Yaskawa INFORM job: OK_R2_O38-47,64(2)(90,0)_MPOK.JBI

/JOB
//NAME OK_R2_O38-47,64(2)(90,0)_MPOK
///FOLDERNAME X4
//POS
///NPOS 359,359,359,19,0,0
///TOOL 0
///POSTYPE PULSE
///PULSE
C00000=102904,-190754,-108658,56793,33718,-43054
C00001=112112,-124440,-79629,37912,40591,-30924
C00002=145621,-43895,-45824,14341,74181,-8322
C00003=153971,-33006,-36006,12070,72386,-5523
C00004=154481,-29919,-31590,11999,71202,-5460
C00005=154481,-29717,-30452,12039,70618,-5519
C00006=154481,-29893,-31438,12004,71123,-5468
C00007=153832,-33137,-33612,12213,70898,-5727
C00008=153832,-32934,-32528,12252,70348,-5784
C00009=153968,-31157,-31341,12198,70507,-5716
C00010=153832,-32934,-32528,12252,70348,-5784
C00011=152546,-38024,-38116,12561,71351,-6144
C00012=150032,-44426,-43245,13273,71622,-7027
C00013=145621,-43895,-45824,14341,74181,-8322
C00014=126188,-124725,-79701,29915,35046,-24780
C00015=102904,-190754,-108658,56793,33718,-43054
C00016=131529,-193853,-113060,37345,24088,-27542
C00017=124211,-86804,-80218,19393,77786,-15538
C00018=164541,26866,21690,9198,66417,-2237
C00019=165950,30734,27944,8880,64418,-1868
C00020=167698,37628,37678,8494,61807,-1405
C00021=167698,38233,39472,8555,61023,-1465
C00022=167698,37628,37678,8494,61807,-1405
C00023=167356,33830,33782,8572,62285,-1498
C00024=167337,34588,35914,8650,61376,-1577
C00025=167338,36654,38036,8669,61135,-1595
C00026=167337,34588,35914,8650,61376,-1577
C00027=169007,24634,18452,7731,66783,-560
C00028=157238,-13932,-14846,11323,68842,-4717
C00029=124389,11727,6427,19504,75270,-15913
C00030=120681,54794,37232,20001,79157,-16624
C00031=120183,64187,51861,20385,75351,-17454
C00032=120121,65987,55496,20510,74134,-17689
C00033=120121,66491,57153,20582,73419,-17815
C00034=120121,65987,55496,20510,74134,-17689
C00035=119196,62638,51610,20616,74997,-17884
C00036=119196,63145,53380,20691,74219,-18021
C00037=119742,65256,55831,20631,73685,-17913
C00038=119196,63145,53380,20691,74219,-18021
C00039=119070,39614,17457,20118,83667,-16456
C00040=118481,-15017,-9678,20946,73127,-18482
C00041=136947,-127922,-100425,-9768,37977,-3776
C00042=166532,-153428,-115250,-33739,42272,11545
C00043=160883,-131526,-133102,3483,78120,6366
C00044=103370,-159686,-136025,1765,64172,8056
C00045=97179,-138237,-129333,10238,76593,-11306
C00046=96065,-128281,-122439,10507,77596,-11607
C00047=96065,-128106,-120653,10546,76604,-11690
C00048=96065,-128281,-122439,10507,77596,-11607
C00049=96974,-121186,-120234,10189,79734,-11117
C00050=96065,-128281,-122439,10507,77596,-11607
C00051=80019,-98046,-111669,14399,88698,-15911
C00052=80077,-97852,-111516,14385,88694,-15892
C00053=80077,-98331,-110658,14385,87944,-15982
C00054=80077,-97897,-111441,14385,88627,-15900
C00055=80867,-94680,-110202,14197,89359,-15553
C00056=80077,-97897,-111441,14385,88627,-15900
C00057=77060,-103837,-123440,15157,93336,-16325
C00058=77104,-103620,-123385,15148,93404,-16303
C00059=82212,-117279,-126602,8714,87753,-18646
C00060=83304,-119533,-127995,7425,87342,-19011
C00061=83304,-120285,-126924,7427,86307,-19072
C00062=83304,-120125,-127175,7427,86540,-19060
C00063=84285,-114583,-125380,7184,88184,-18645
C00064=83304,-120125,-127175,7427,86540,-19060
C00065=78124,-131037,-133000,8681,85036,-20864
C00066=78124,-131037,-133000,8681,85036,-20864
C00067=80781,-132367,-131851,8063,83392,-20088
C00068=80781,-132658,-130737,8071,82565,-20142
C00069=80781,-132579,-131090,8068,82820,-20125
C00070=82215,-124520,-128659,7695,85306,-19491
C00071=80136,-136061,-133167,8229,82377,-20371
C00072=80218,-134686,-135534,8183,84509,-20204
C00073=75563,-118157,-129697,13391,92336,-27261
C00074=84024,-123631,-127734,11595,87159,-24981
C00075=84024,-123979,-126960,11598,86516,-25042
C00076=84024,-123746,-127494,11596,86956,-25000
C00077=85048,-122093,-126977,11373,87337,-24623
C00078=81994,-135324,-132084,12059,84184,-25946
C00079=81994,-133752,-136174,12028,87438,-25630
C00080=81994,-133752,-136174,12028,87438,-25630
C00081=83107,-120864,-125937,11789,87596,-25245
C00082=83880,-119254,-122492,11630,86222,-25116
C00083=83880,-119583,-121326,11637,85351,-25197
C00084=83880,-119399,-122020,11633,85865,-25149
C00085=85062,-113328,-120022,11369,87556,-24598
C00086=83880,-119399,-122020,11633,85865,-25149
C00087=83464,-119333,-123502,11716,86850,-25194
C00088=84085,-116294,-122008,11580,87393,-24935
C00089=84085,-116863,-120480,11583,86184,-25047
C00090=84085,-116689,-121008,11580,86590,-25010
C00091=85140,-111307,-119205,11348,88071,-24523
C00092=84085,-116194,-122230,11576,87577,-24918
C00093=82864,-118268,-130611,11862,91757,-24924
C00094=82864,-118268,-130611,11862,91757,-24924
C00095=86851,-110557,-120071,10968,88745,-23893
C00096=86851,-111341,-118540,10968,87421,-24011
C00097=86851,-110811,-119621,10968,88345,-23929
C00098=88598,-109546,-119189,10575,88500,-23337
C00099=86851,-110811,-119621,10968,88345,-23929
C00100=83825,-124590,-131318,11630,88867,-24881
C00101=82909,-127853,-136097,11834,90233,-25054
C00102=84148,-125178,-125504,11579,85018,-25131
C00103=81186,-118241,-121828,12198,86718,-25964
C00104=81186,-118533,-120824,12201,85966,-26037
C00105=81186,-118483,-121017,12200,86107,-26023
C00106=82314,-113243,-119285,11952,87535,-25506
C00107=81186,-118241,-121828,12198,86718,-25964
C00108=87931,-140644,-131144,10841,80108,-24284
C00109=89960,-139833,-128047,10433,78377,-23732
C00110=89960,-139550,-127065,10448,77925,-23770
C00111=89960,-139622,-127307,10444,78035,-23761
C00112=90753,-134395,-125809,10209,79670,-23349
C00113=89456,-143397,-129529,10578,77538,-23979
C00114=95203,-107502,-133483,6717,98684,-21003
C00115=95203,-107502,-133483,6717,98684,-21003
C00116=-70091,-137861,-134613,-19540,89589,11549
C00117=-70091,-137861,-134613,-19540,89589,11549
C00118=-89914,-142582,-130695,-14485,81723,10120
C00119=-90202,-137048,-128128,-14398,82897,9883
C00120=-90202,-136718,-126391,-14423,82025,9985
C00121=-90202,-136862,-127082,-14413,82365,9945
C00122=-91010,-131454,-125503,-14223,83978,9478
C00123=-90202,-137070,-128271,-14397,82970,9874
C00124=-76195,-137070,-128271,-14397,82970,9874
C00125=-74994,-123934,-123423,-14560,86840,9835
C00126=-74994,-124092,-122198,-14564,86029,9931
C00127=-74994,-124005,-122955,-14561,86525,9872
C00128=-76141,-119465,-121513,-14342,87728,9340
C00129=-72631,-133219,-128550,-14998,85696,10781
C00130=-72631,-131663,-134232,-14989,89852,10278
C00131=-50716,-132590,-134806,-14983,95067,21778
C00132=-53786,-122460,-125023,-14607,93736,20890
C00133=-54881,-121663,-124068,-14472,93371,20558
C00134=-54881,-122014,-122728,-14450,92397,20672
C00135=-54881,-121856,-123398,-14460,92875,20616
C00136=-56721,-117465,-121986,-14267,93906,19868
C00137=-54881,-121856,-123398,-14460,92875,20616
C00138=-55322,-120745,-123309,-14420,93300,20415
C00139=-55322,-120747,-123302,-14420,93295,20416
C00140=-55322,-120978,-122461,-14407,92679,20487
C00141=-55322,-120864,-122902,-14414,92999,20450
C00142=-56710,-117554,-121835,-14266,93775,19889
C00143=-54436,-122887,-123768,-14509,92662,20793
C00144=-54436,-122067,-126198,-14556,94519,20574
C00145=-53688,-126302,-127242,-14482,93230,21000
C00146=-7968,-117738,-135568,-14910,102458,19890
C00147=-7968,-117738,-135568,-14910,102458,19890
C00148=-4119,-116606,-125698,-15061,97809,21757
C00149=-7770,-114903,-122318,-14590,96007,20739
C00150=-7770,-115418,-121244,-14557,95111,20843
C00151=-7770,-115024,-122084,-14598,95810,20761
C00152=-9375,-110655,-120613,-14452,96836,20097
C00153=-7770,-115024,-122084,-14598,95810,20761
C00154=-10569,-102485,-118509,-17167,107955,30726
C00155=-17135,-102893,-117262,-17068,107079,30955
C00156=121481,-92648,-105286,5369,115019,86755
C00157=120615,-96829,-107734,5213,114434,86412
C00158=-23859,-150611,-131722,-11614,81196,13147
C00159=-6314,-100679,-115153,-9004,91229,18831
C00160=-5878,-99274,-114584,-9040,91548,18958
C00161=-5881,-109040,-123705,-8960,92007,18939
C00162=-6434,-120006,-133010,-8839,92040,18760
C00163=12667,-120051,-129788,19636,91452,-63850
C00164=15640,-171133,-136982,20070,70138,-66271
C00165=-3139,-164995,-126377,36529,73517,-73495
C00166=120436,-95190,-80290,14692,43277,-16053
C00167=119715,-95468,-78930,15521,42464,-16563
C00168=-536,-140958,-118488,38156,78150,-70805
C00169=15896,-141744,-117960,35334,65109,-67636
C00170=22809,-140005,-116746,30747,58039,-62654
C00171=24043,-118481,-124771,21586,79008,-61529
C00172=24043,-118481,-124771,21586,79008,-61529
C00173=75030,-118005,-124618,21594,79160,-61521
C00174=115715,-153549,-128562,-15788,54400,-49074
C00175=122128,-153495,-122411,-24310,49621,-45021
C00176=120438,-96789,-101713,1489,48968,-3516
C00177=120356,-99154,-104149,1548,49253,-3547
C00178=84431,-115837,-110938,-1908,55230,-61215
C00179=103640,-112319,-105648,-32381,57576,-46168
C00180=90828,-138253,-118809,-13315,45388,-56216
C00181=90828,-138253,-118809,-13315,45388,-56216
C00182=90828,-142934,-129815,-12421,49655,-56806
C00183=90829,-142933,-129813,-12421,49658,-56806
C00184=119872,-163920,-132846,-33283,49576,-42941
C00185=126809,-145866,-124115,-34845,55617,-41735
C00186=120835,-94912,-106201,-4597,84031,-3620
C00187=120296,-100536,-106811,-4468,81494,-3706
C00188=119927,-142522,-122915,-31276,53757,-44413
C00189=77611,-97741,-105288,-5509,51883,-63151
C00190=72401,-92495,-101825,-908,50569,-65138
C00191=77718,-122737,-116129,-5642,44048,-62545
C00192=53268,-154266,-130714,22807,48565,-72872
C00193=53268,-154266,-130714,22807,48565,-72872
C00194=65704,-162398,-123942,17029,37659,-69009
C00195=71918,-162932,-118398,17522,29983,-67437
C00196=120621,-91661,-79831,-4809,93096,80691
C00197=120610,-95504,-82099,-4805,92519,80709
C00198=65560,-150384,-115443,21255,35856,-69819
C00199=55757,-109501,-106397,19317,55331,-70255
C00200=57003,-110782,-106224,17216,52464,-70603
C00201=59740,-113209,-105691,12878,47416,-70775
C00202=50265,-141050,-116073,27906,38980,-77613
C00203=41790,-175398,-134696,41509,59591,-72504
C00204=40096,-167295,-132799,40833,62675,-71982
C00205=66233,-176056,-134792,18069,45461,-58242
C00206=120613,-98309,-97516,18774,58387,-20033
C00207=120296,-100165,-96633,19249,57041,-20409
C00208=66115,-175766,-134726,18105,45590,-58274
C00209=64821,-169609,-132859,18260,47793,-58447
C00210=52681,-139177,-124950,28110,65688,-66537
C00211=50721,-103471,-113434,27126,76369,-64663
C00212=50688,-103205,-113338,27131,76448,-64657
C00213=56284,-114059,-116499,20977,66017,-65546
C00214=54527,-104423,-113142,21374,69156,-65613
C00215=49750,-132075,-132074,23871,68057,-67633
C00216=51888,-141517,-135531,28423,71943,-65142
C00217=58410,-142164,-121837,32385,67064,-69630
C00218=59671,-133628,-117738,33640,70981,-70965
C00219=120621,-92022,-79948,5717,93324,87803
C00220=120611,-95871,-82213,5711,92744,87773
C00221=92104,-176981,-128268,-2909,38154,-41832
C00222=76594,-127084,-115767,-3536,56171,-41355
C00223=99425,-103206,-107694,-29386,75495,-21963
C00224=100715,-115554,-120696,-29641,77391,-21955
C00225=99511,-125054,-130815,-29118,78165,-22610
C00226=-30978,-142903,-136378,-16839,87530,25088
C00227=-49033,-141162,-127974,-10600,82449,19659
C00228=120514,-92773,-72492,-63824,26217,40707
C00229=122096,-91517,-72885,-63277,27653,40461
C00230=-46723,-132150,-125263,-10235,84639,20316
C00231=-38144,-96146,-111322,-6693,87070,23612
C00232=-37356,-92674,-109966,-6904,88077,23811
C00233=-38688,-150385,-135608,-6755,74185,24124
C00234=-34744,-121097,-133452,-9828,92546,23976
C00235=-92930,-150385,-135608,-6755,74185,24124
C00236=-108565,-138971,-125572,-2320,72996,18698
C00237=120610,-93305,-77258,-53115,31058,-22991
C00238=120294,-94166,-75974,-54567,30127,-22239
C00239=-116035,-135916,-124846,7405,75208,6894
C00240=-75325,-100736,-113015,-4102,85156,20630
C00241=-87779,-91378,-109906,9606,90211,4845
C00242=-92139,-118134,-128268,12138,88585,1394
C00243=-96790,-150711,-134355,17072,70659,-2161
C00244=-96790,-150711,-134355,17072,70659,-2161
C00245=-652,-114254,-134536,4800,91191,3391
C00246=166532,-153428,-115250,-33739,42272,11545
C00247=166532,-153428,-115250,-33739,42272,11545
C00248=124114,-84683,-61597,48557,28871,52530
C00249=120971,1491,10647,53300,28999,53238
C00250=122160,19295,36771,64461,24491,47841
C00251=122378,23552,43589,68524,23503,45877
C00252=120673,10502,19535,54974,28515,52685
C00253=120213,7916,15945,54003,29309,53162
C00254=117639,31595,51593,71855,26327,43764
C00255=117542,21645,38109,65998,27616,46690
C00256=116582,-33548,-30911,47449,36332,56383
C00257=108749,-129529,-72544,82443,35289,33776
C00258=107659,-149780,-91003,80990,36184,34408
C00259=234701,-24447,-54419,-57638,71697,-57534
C00260=192045,-4471,-49137,-31395,56880,-70337
C00261=158835,26744,-30866,6797,89214,-71249
C00262=162394,21957,-27190,-640,114363,-79561
C00263=164064,23195,-19161,-1804,117838,-80318
C00264=164490,20804,-18265,-1733,116068,-80136
C00265=164232,27876,-3751,-4961,127378,-83177
C00266=164200,29818,-583,-4904,126429,-83142
C00267=163648,20652,-18364,-1809,116035,-80437
C00268=163648,20933,-18885,-1817,116499,-80445
C00269=162721,21060,-18767,-1901,116472,-80776
C00270=162825,20781,-18263,-1883,116024,-80730
C00271=161869,20798,-18246,-1969,116003,-81071
C00272=161869,21389,-19316,-1987,116965,-81088
C00273=162128,7432,-36637,578,111538,-80469
C00274=155887,-31466,-65010,7215,96475,-81562
C00275=162590,-38859,-73812,1668,81223,-78508
C00276=179792,32070,-16354,-13350,79915,-65662
C00277=186878,-39073,-38836,-41246,34970,-63358
C00278=187458,-25431,-34231,-31791,43871,-67525
C00279=188256,-32514,-32154,-43117,35074,-62369
C00280=188651,-34827,-34931,-42941,35654,-62475
C00281=186634,-25994,-34626,-31183,43526,-67848
C00282=186634,-26042,-35404,-30940,43918,-67999
C00283=179776,-30769,-38597,-15117,38446,-76230
C00284=179862,-30379,-37602,-15341,38064,-76107
C00285=178691,-31104,-38049,-14184,37759,-76698
C00286=185299,-29135,-41036,-26782,46455,-69327
C00287=188726,-40923,-42933,-41373,37038,-63352
C00288=196569,5763,-30645,-36969,53415,-67065
C00289=234701,-24447,-54419,-57638,71697,-57534
C00290=149956,-140196,-108889,10254,17658,75195
C00291=133880,-29999,-59672,20958,46846,70848
C00292=133880,-29999,-59672,20958,46846,70848
C00293=122391,19095,38576,70751,31293,46770
C00294=123405,34197,53895,59777,34432,53030
C00295=120673,9158,15746,60306,37604,52768
C00296=120213,7880,15913,61361,37506,52152
C00297=128224,26945,46555,56859,32016,55120
C00298=125984,18051,32799,53129,35607,56921
C00299=127465,-31665,-25778,42614,42048,63033
C00300=111364,-124873,-96714,53393,47795,55834
C00301=154186,-159927,-117173,847,12331,79725
C00302=85861,-99082,-105113,44329,59147,50836
C00303=83984,-106882,-107996,46165,58479,49488
C00304=120674,-14372,-36148,15341,86455,69375
C00305=120676,-10921,-33498,15340,86592,69392
C00306=125651,22057,-6379,9907,105287,72561
C00307=121175,-12454,-34682,15229,86445,69544
C00308=120675,-14159,-37235,15335,87207,69469
C00309=127950,19387,-8926,9965,105208,73352
C00310=120676,-11639,-34054,15340,86566,69391
C00311=120674,-14390,-36162,15341,86455,69375
C00312=120676,-14354,-36134,15765,85734,-14225
C00313=120676,-14354,-36134,15765,85734,-14225
C00314=121459,-13803,-34784,15590,85060,-14040
C00315=120676,-14158,-37234,15757,86484,-14129
C00316=120165,-16255,-37568,15883,85739,-14397
C00317=124003,-16979,-37218,14998,84465,-13252
C00318=120676,-14374,-36149,15765,85733,-14224
C00319=120676,-14373,-36148,15765,85733,-14225
C00320=98406,-95981,-107671,30899,65126,-25478
C00321=97498,-103141,-110365,31836,63713,-26282
C00322=97498,-103141,-110365,31836,63713,-26282
C00323=151185,-64492,-56891,27025,41971,76525
C00324=173123,2305,9538,10200,51383,-14399
C00325=173123,2305,9538,10200,51383,-14399
C00326=174903,14820,25056,9713,48090,-13953
C00327=177435,27097,40637,4614,49072,-8771
C00328=187315,39588,15664,-2886,77004,-72543
C00329=187570,37474,12233,-2951,78037,-72481
C00330=182393,31000,44587,2257,48438,-6634
C00331=178652,16834,25077,3801,53300,-8079
C00332=172335,1396,7152,6372,56784,-10488
C00333=165460,10359,17772,9398,55625,-13216
C00334=160953,16615,26241,11506,54240,-15214
C00335=161039,26979,37798,10163,56196,-14889
C00336=187825,35310,11263,-3318,76749,7758
C00337=187564,37491,12251,-3232,77251,7657
C00338=166034,27602,38530,8404,55496,-12935
C00339=166237,17707,23738,7975,59455,-12552
C00340=164665,16592,22700,-1550,58461,-2398
C00341=168038,24831,35842,-7675,55527,4086
C00342=167355,24747,35761,-7424,55472,3814
C00343=168052,14770,21803,-7392,58972,3848
C00344=169021,11489,3544,7471,65997,66244
C00345=151185,-64492,-56891,27025,41971,76525
C00346=139846,-133648,-87236,40448,26560,70293
C00347=136335,-97157,-88666,6240,65884,69249
C00348=141826,-62430,-72987,3929,73707,71532
C00349=140052,-21130,-52867,-24635,78479,75610
C00350=128083,45376,-375,-18819,101882,68514
C00351=126763,43366,-45,-18530,100432,68297
C00352=126966,41908,238,-18497,99599,68497
C00353=135984,107314,69748,-14048,119719,69614
C00354=135785,103774,66356,-14147,119946,69504
C00355=122863,47542,6419,-17829,97882,67372
C00356=124413,47820,3838,-18170,99852,67599
C00357=123183,-7178,-53151,6497,97844,73056
C00358=89230,-40025,-45988,57168,55507,51535
BC00000=155259,430035,251707
BC00001=155259,370518,251707
BC00002=155259,370518,251707
BC00003=155259,370518,251707
BC00004=155259,370518,251707
BC00005=155259,370518,251707
BC00006=155259,370518,251707
BC00007=155259,370518,251707
BC00008=155259,370518,251707
BC00009=155259,370518,251707
BC00010=155259,370518,251707
BC00011=155259,370518,251707
BC00012=155259,370518,251707
BC00013=155259,370518,251707
BC00014=155259,370518,251707
BC00015=155259,430035,251707
BC00016=334621,427363,453529
BC00017=334621,347923,356901
BC00018=334621,347923,326221
BC00019=334621,347923,326221
BC00020=334621,347923,326221
BC00021=334621,347923,326221
BC00022=334621,347923,326221
BC00023=334621,347923,326221
BC00024=334621,347923,326221
BC00025=334621,347923,326221
BC00026=334621,347923,326221
BC00027=334621,347923,326221
BC00028=334621,347923,326221
BC00029=334621,347923,326221
BC00030=324461,347923,240729
BC00031=324461,347923,240729
BC00032=324461,347923,240729
BC00033=324461,347923,240729
BC00034=324461,347923,240729
BC00035=324461,347923,240729
BC00036=324461,347923,240729
BC00037=324461,347923,240729
BC00038=324461,347923,240729
BC00039=324461,347923,240729
BC00040=324461,347923,382261
BC00041=343276,399368,267274
BC00042=343276,522663,1074774
BC00043=343276,475512,1074774
BC00044=343276,247728,1074774
BC00045=336018,234000,1074774
BC00046=336018,234000,1074774
BC00047=336018,234000,1074774
BC00048=336018,234000,1074774
BC00049=336018,234000,1074774
BC00050=336018,234000,1074774
BC00051=336018,234000,1074774
BC00052=336018,234000,1074774
BC00053=336018,234000,1074774
BC00054=336018,234000,1074774
BC00055=336018,234000,1074774
BC00056=336018,234000,1074774
BC00057=336018,234000,1074774
BC00058=371484,186454,1072332
BC00059=371484,178806,1072332
BC00060=371484,177238,1072332
BC00061=371484,177238,1072332
BC00062=371484,177238,1072332
BC00063=371484,177238,1072332
BC00064=371484,177238,1072332
BC00065=371484,177238,1072332
BC00066=310125,182966,1071793
BC00067=310125,182966,1071793
BC00068=310125,182966,1071793
BC00069=310125,182966,1071793
BC00070=310125,182966,1071793
BC00071=310125,182966,1071793
BC00072=310125,182966,1071793
BC00073=246912,213302,1071793
BC00074=246912,213302,1071793
BC00075=246912,213302,1071793
BC00076=246912,213302,1071793
BC00077=246912,213302,1071793
BC00078=246912,213302,1071793
BC00079=246912,213302,1071793
BC00080=143996,226029,1063218
BC00081=143996,226029,1063218
BC00082=143996,226029,1063218
BC00083=143996,226029,1063218
BC00084=143996,226029,1063218
BC00085=143996,226029,1063218
BC00086=143996,226029,1063218
BC00087=107402,233101,1063218
BC00088=107402,233101,1063218
BC00089=107402,233101,1063218
BC00090=107402,233101,1063218
BC00091=107402,233101,1063218
BC00092=107402,233101,1063218
BC00093=107402,233101,1063218
BC00094=126000,290967,1063218
BC00095=126000,290967,1063218
BC00096=126000,290967,1063218
BC00097=126000,290967,1063218
BC00098=126000,290967,1063218
BC00099=126000,290967,1063218
BC00100=126000,290967,1063218
BC00101=32367,290967,1063218
BC00102=33707,241035,1063218
BC00103=33707,241035,1063218
BC00104=33707,241035,1063218
BC00105=33707,241035,1063218
BC00106=33707,241035,1063218
BC00107=33707,241035,1063218
BC00108=7031,245739,1063218
BC00109=6955,243723,1064247
BC00110=6955,243723,1064247
BC00111=6955,243723,1064247
BC00112=6955,243723,1064247
BC00113=6955,243723,1064247
BC00114=6955,243723,1064247
BC00115=25087,359545,1064247
BC00116=1824,213285,1064247
BC00117=1824,167485,1064247
BC00118=1824,167485,1064247
BC00119=1824,167485,1064247
BC00120=1824,167485,1064247
BC00121=1824,167485,1064247
BC00122=1824,167485,1064247
BC00123=1824,167485,1064247
BC00124=32224,168989,1065766
BC00125=32224,168989,1065766
BC00126=32224,168989,1065766
BC00127=32224,168989,1065766
BC00128=32224,168989,1065766
BC00129=32224,168989,1065766
BC00130=32224,168989,1065766
BC00131=75962,188381,1065766
BC00132=75961,188380,1065763
BC00133=75961,188380,1065763
BC00134=75961,188380,1065763
BC00135=75961,188380,1065763
BC00136=75961,188380,1065763
BC00137=75961,188380,1065763
BC00138=117533,188380,1065763
BC00139=117533,188380,1065763
BC00140=117533,188380,1065763
BC00141=117533,188380,1065763
BC00142=117533,188380,1065763
BC00143=117533,188380,1065763
BC00144=117533,188380,1065763
BC00145=56658,153797,1065859
BC00146=56658,153797,1065859
BC00147=30873,87130,1065859
BC00148=45198,87130,1065859
BC00149=45198,87130,1065859
BC00150=45198,87130,1065859
BC00151=45198,87131,1065856
BC00152=45198,87131,1065856
BC00153=45198,87131,1065856
BC00154=45198,87131,1065853
BC00155=45198,87131,1065852
BC00156=145241,272408,1075139
BC00157=145241,272408,1075139
BC00158=45198,87131,1065851
BC00159=45198,87131,1065851
BC00160=45198,87131,1065851
BC00161=45198,87131,1065851
BC00162=45198,87131,1065851
BC00163=50333,237173,1065851
BC00164=50333,237173,1065851
BC00165=50333,237173,1065851
BC00166=156919,411124,1075139
BC00167=156919,411124,1075139
BC00168=50333,237173,1065851
BC00169=72120,237173,1065851
BC00170=72120,237173,1065851
BC00171=72120,237173,1065851
BC00172=58630,250517,1065851
BC00173=17,309807,1065851
BC00174=17,261367,1065849
BC00175=17,261367,1065849
BC00176=369303,316629,1075139
BC00177=369303,316629,1075139
BC00178=17,261367,1065849
BC00179=17,261367,1065849
BC00180=17,261367,1065849
BC00181=17,263287,1072219
BC00182=17,340739,1070027
BC00183=271547,213230,1070026
BC00184=312655,207246,1064979
BC00185=312655,207246,1064979
BC00186=4070,330706,1075139
BC00187=4070,330706,1075139
BC00188=312655,207246,1064979
BC00189=312655,207246,1064979
BC00190=312655,207246,1064979
BC00191=312655,207246,1064979
BC00192=312655,207246,1064979
BC00193=280580,230258,1064979
BC00194=280580,230258,1064979
BC00195=280580,230258,1064979
BC00196=125976,418809,1075139
BC00197=125976,418809,1075139
BC00198=280580,230258,1064979
BC00199=280580,230258,1064976
BC00200=280580,230258,1064977
BC00201=280581,230257,1064979
BC00202=280580,230258,1064979
BC00203=280580,230258,1064979
BC00204=211671,216434,1064979
BC00205=204230,216434,1064979
BC00206=168817,338507,1075139
BC00207=168817,338507,1075139
BC00208=204230,216434,1064979
BC00209=204230,216434,1064979
BC00210=204230,216434,1064979
BC00211=204230,216434,1064979
BC00212=204230,216434,1064979
BC00213=204230,216434,1064979
BC00214=204230,216434,1064979
BC00215=204230,216434,1064979
BC00216=93787,231658,1064979
BC00217=93787,231658,1064979
BC00218=93788,231658,1064978
BC00219=27652,419064,1075139
BC00220=27652,419064,1075139
BC00221=93788,231658,1064978
BC00222=93788,231658,1064978
BC00223=93788,231658,1064978
BC00224=93788,231658,1064978
BC00225=93788,231658,1064978
BC00226=58883,202583,1068082
BC00227=58883,202583,1068082
BC00228=345487,351087,1075139
BC00229=345487,351087,1075139
BC00230=58883,202583,1068082
BC00231=58883,202583,1068082
BC00232=58883,202583,1068082
BC00233=58883,202583,1068082
BC00234=58123,202583,1068180
BC00235=1968,161247,1068082
BC00236=1968,161247,1068082
BC00237=310134,354281,1075139
BC00238=310134,354281,1075139
BC00239=1968,161247,1068082
BC00240=1968,161247,1068082
BC00241=1968,161247,1068082
BC00242=1968,161247,1068082
BC00243=1968,161247,1068082
BC00244=1968,356313,1068082
BC00245=56320,430883,1064743
BC00246=343276,475512,1074774
BC00247=343276,475512,418626
BC00248=326702,360123,309424
BC00249=326065,355687,311834
BC00250=325331,353932,278401
BC00251=325331,353932,278401
BC00252=322890,348232,200536
BC00253=322890,348232,200536
BC00254=325331,353932,278401
BC00255=325331,353932,278401
BC00256=325331,353932,278401
BC00257=326702,394520,413552
BC00258=326702,482298,413552
BC00259=301892,455031,17
BC00260=301892,455031,17
BC00261=209904,428615,17
BC00262=165530,382080,91459
BC00263=159566,375826,103748
BC00264=159566,375826,103748
BC00265=146818,362457,130017
BC00266=146818,362457,130017
BC00267=159566,375826,103748
BC00268=159566,375826,103748
BC00269=159566,375826,103748
BC00270=159566,375826,103748
BC00271=159566,375826,103748
BC00272=159566,375826,103748
BC00273=159566,375826,103748
BC00274=160331,376239,102936
BC00275=179623,386657,82465
BC00276=243106,413945,27916
BC00277=213965,383877,85097
BC00278=213965,383877,85097
BC00279=213965,383877,85097
BC00280=213965,383877,85097
BC00281=213965,383877,85097
BC00282=213965,383877,85097
BC00283=213965,383877,85097
BC00284=213965,383877,85097
BC00285=213965,383877,85097
BC00286=213965,383877,85097
BC00287=213965,383877,85097
BC00288=301892,455031,17
BC00289=301892,455031,17
BC00290=376045,502685,343368
BC00291=326979,388611,268695
BC00292=326979,388611,268695
BC00293=314569,362038,322228
BC00294=314569,362038,322228
BC00295=310726,355002,200377
BC00296=310726,355002,200377
BC00297=314569,362038,322228
BC00298=314569,362038,322228
BC00299=314569,362038,322228
BC00300=314569,409194,450098
BC00301=326003,483358,319355
BC00302=108142,501291,133069
BC00303=94929,415794,32572
BC00304=131923,388713,210323
BC00305=131318,389042,183541
BC00306=131077,389173,172829
BC00307=131077,389173,172829
BC00308=131077,389173,172829
BC00309=131077,389173,172829
BC00310=125260,392440,183541
BC00311=125864,392111,210322
BC00312=132288,390101,176526
BC00313=128864,385756,157610
BC00314=127495,384018,150044
BC00315=127495,384018,150044
BC00316=127495,384018,150044
BC00317=127495,384018,150044
BC00318=122392,389386,157610
BC00319=125816,393731,176526
BC00320=132288,412747,17
BC00321=132288,502680,17
BC00322=329813,502680,230019
BC00323=341603,346180,231132
BC00324=341603,346182,356182
BC00325=319069,341990,356182
BC00326=319069,341990,356182
BC00327=319069,341990,385359
BC00328=340757,346640,193638
BC00329=340757,346640,193638
BC00330=319069,341990,385359
BC00331=319069,341990,385359
BC00332=319069,341990,385359
BC00333=319464,342064,382925
BC00334=319464,342064,382925
BC00335=319464,342064,382925
BC00336=344822,337105,170856
BC00337=344822,337105,170856
BC00338=319464,342064,382925
BC00339=319464,342064,382925
BC00340=319464,342064,382925
BC00341=319464,342064,382925
BC00342=319464,342064,382925
BC00343=319464,342064,382925
BC00344=325489,344287,327316
BC00345=341603,346180,395974
BC00346=341603,460199,530170
BC00347=190885,461337,170893
BC00348=190885,404072,170893
BC00349=164847,397070,131538
BC00350=148987,398107,68956
BC00351=148987,398107,68956
BC00352=148987,398107,68956
BC00353=192995,397070,17
BC00354=192995,397070,17
BC00355=148987,398107,68956
BC00356=148987,398107,68956
BC00357=146579,399402,81875
BC00358=106846,403091,165317
EC00000=-798156,-183832
EC00001=-798156,-183832
EC00002=-798156,-183832
EC00003=-798156,-183832
EC00004=-798156,-183832
EC00005=-798156,-183832
EC00006=-798156,-183832
EC00007=-798156,-183832
EC00008=-798156,-183832
EC00009=-798156,-183832
EC00010=-798156,-183832
EC00011=-798156,-183832
EC00012=-798156,-183832
EC00013=-798156,-183832
EC00014=-798156,-183832
EC00015=-798156,-183832
EC00016=-798156,-183832
EC00017=-798156,-183832
EC00018=-798156,-183832
EC00019=-798156,-183832
EC00020=-798156,-183832
EC00021=-798156,-183832
EC00022=-798156,-183832
EC00023=-798156,-183832
EC00024=-798156,-183832
EC00025=-798156,-183832
EC00026=-798156,-183832
EC00027=-798156,-183832
EC00028=-798156,-183832
EC00029=-798156,-183832
EC00030=-798156,-183832
EC00031=-798156,-183832
EC00032=-798156,-183832
EC00033=-798156,-183832
EC00034=-798156,-183832
EC00035=-798156,-183832
EC00036=-798156,-183832
EC00037=-798156,-183832
EC00038=-798156,-183832
EC00039=-798156,-183832
EC00040=-798156,-183832
EC00041=-798156,-183832
EC00042=-798156,-183832
EC00043=-798156,-183832
EC00044=-798156,-183832
EC00045=-798156,-183832
EC00046=-798156,-183832
EC00047=-798156,-183832
EC00048=-798156,-183832
EC00049=-798156,-183832
EC00050=-798156,-183832
EC00051=-798156,-183832
EC00052=-798156,-183832
EC00053=-798156,-183832
EC00054=-798156,-183832
EC00055=-798156,-183832
EC00056=-798156,-183832
EC00057=-798156,-183832
EC00058=-798156,-183832
EC00059=-798156,-183832
EC00060=-798156,-183832
EC00061=-798156,-183832
EC00062=-798156,-183832
EC00063=-798156,-183832
EC00064=-798156,-183832
EC00065=-798156,-183832
EC00066=-798156,-183832
EC00067=-798156,-183832
EC00068=-798156,-183832
EC00069=-798156,-183832
EC00070=-798156,-183832
EC00071=-798156,-183832
EC00072=-798156,-183832
EC00073=-798156,-183832
EC00074=-798156,-183832
EC00075=-798156,-183832
EC00076=-798156,-183832
EC00077=-798156,-183832
EC00078=-798156,-183832
EC00079=-798156,-183832
EC00080=-798156,-183832
EC00081=-798156,-183832
EC00082=-798156,-183832
EC00083=-798156,-183832
EC00084=-798156,-183832
EC00085=-798156,-183832
EC00086=-798156,-183832
EC00087=-798156,-183832
EC00088=-798156,-183832
EC00089=-798156,-183832
EC00090=-798156,-183832
EC00091=-798156,-183832
EC00092=-798156,-183832
EC00093=-798156,-183832
EC00094=-798156,-183832
EC00095=-798156,-183832
EC00096=-798156,-183832
EC00097=-798156,-183832
EC00098=-798156,-183832
EC00099=-798156,-183832
EC00100=-798156,-183832
EC00101=-798156,-183832
EC00102=-798156,-183832
EC00103=-798156,-183832
EC00104=-798156,-183832
EC00105=-798156,-183832
EC00106=-798156,-183832
EC00107=-798156,-183832
EC00108=-798156,-183832
EC00109=-798156,-183832
EC00110=-798156,-183832
EC00111=-798156,-183832
EC00112=-798156,-183832
EC00113=-798156,-183832
EC00114=-798156,-183832
EC00115=-798156,-183832
EC00116=-798156,-183832
EC00117=-798156,-183832
EC00118=-798156,-183832
EC00119=-798156,-183832
EC00120=-798156,-183832
EC00121=-798156,-183832
EC00122=-798156,-183832
EC00123=-798156,-183832
EC00124=-798156,-183832
EC00125=-798156,-183832
EC00126=-798156,-183832
EC00127=-798156,-183832
EC00128=-798156,-183832
EC00129=-798156,-183832
EC00130=-798156,-183832
EC00131=-798156,-183832
EC00132=-798154,-183832
EC00133=-798154,-183832
EC00134=-798154,-183832
EC00135=-798154,-183832
EC00136=-798154,-183832
EC00137=-798154,-183832
EC00138=-798154,-183832
EC00139=-798154,-183832
EC00140=-798154,-183832
EC00141=-798154,-183832
EC00142=-798154,-183832
EC00143=-798154,-183832
EC00144=-798154,-183832
EC00145=-799965,-183832
EC00146=-799965,-183832
EC00147=-799965,-183832
EC00148=-799965,-183832
EC00149=-799965,-183832
EC00150=-799965,-183832
EC00151=-799962,-183833
EC00152=-799962,-183833
EC00153=-799962,-183833
EC00154=-799960,-183834
EC00155=-799958,-183835
EC00156=-975524,-183832
EC00157=-975524,-183832
EC00158=-799958,-183834
EC00159=-799958,-183834
EC00160=-799958,-183834
EC00161=-799958,-183834
EC00162=-799958,-183834
EC00163=-799958,-183834
EC00164=-799958,-183834
EC00165=-799958,-183834
EC00166=-975524,-183832
EC00167=-975524,-183832
EC00168=-799958,-183834
EC00169=-799958,-183834
EC00170=-799958,-183834
EC00171=-799958,-183834
EC00172=-799958,-183834
EC00173=-799958,-183834
EC00174=-799955,-183834
EC00175=-799955,-183834
EC00176=-975524,-183832
EC00177=-975524,-183832
EC00178=-799955,-183834
EC00179=-799955,-183834
EC00180=-799955,-183834
EC00181=-799955,-183834
EC00182=-799954,-183835
EC00183=-799951,-183835
EC00184=-799951,-183835
EC00185=-799951,-183835
EC00186=-975524,-183832
EC00187=-975524,-183832
EC00188=-799951,-183835
EC00189=-799951,-183835
EC00190=-799951,-183835
EC00191=-799951,-183835
EC00192=-799951,-183835
EC00193=-799951,-183835
EC00194=-799951,-183835
EC00195=-799951,-183835
EC00196=-975524,-183832
EC00197=-975524,-183832
EC00198=-799951,-183835
EC00199=-799949,-183836
EC00200=-799950,-183836
EC00201=-799948,-183837
EC00202=-799951,-183835
EC00203=-799951,-183835
EC00204=-799951,-183835
EC00205=-799951,-183835
EC00206=-975524,-183832
EC00207=-975524,-183832
EC00208=-799951,-183835
EC00209=-799951,-183835
EC00210=-799951,-183835
EC00211=-799951,-183835
EC00212=-799951,-183835
EC00213=-799951,-183835
EC00214=-799951,-183835
EC00215=-799951,-183835
EC00216=-799951,-183835
EC00217=-799951,-183835
EC00218=-799949,-183835
EC00219=-975524,-183832
EC00220=-975524,-183832
EC00221=-799949,-183835
EC00222=-799949,-183835
EC00223=-799949,-183835
EC00224=-799949,-183835
EC00225=-799949,-183835
EC00226=-799949,-183835
EC00227=-799949,-183835
EC00228=-975524,-183832
EC00229=-975524,-183832
EC00230=-799949,-183835
EC00231=-799949,-183835
EC00232=-799949,-183835
EC00233=-799949,-183835
EC00234=-799949,-183835
EC00235=-799949,-183835
EC00236=-799949,-183835
EC00237=-975524,-183832
EC00238=-975524,-183832
EC00239=-799949,-183835
EC00240=-799949,-183835
EC00241=-799949,-183835
EC00242=-799949,-183835
EC00243=-799949,-183835
EC00244=-799949,-183835
EC00245=-802129,-183835
EC00246=-798156,-183832
EC00247=-798156,-183832
EC00248=-798156,-183832
EC00249=-798156,-183832
EC00250=-798154,-183835
EC00251=-798154,-183835
EC00252=-798156,-183832
EC00253=-798156,-183832
EC00254=-798154,-183835
EC00255=-798154,-183835
EC00256=-798154,-183835
EC00257=-798156,-183832
EC00258=-798156,-183832
EC00259=-798156,-183832
EC00260=-798156,-183832
EC00261=-798156,-183832
EC00262=-798156,-183832
EC00263=-798156,-183832
EC00264=-798156,-183832
EC00265=-798156,-183832
EC00266=-798156,-183832
EC00267=-798156,-183832
EC00268=-798156,-183832
EC00269=-798156,-183832
EC00270=-798156,-183832
EC00271=-798156,-183832
EC00272=-798156,-183832
EC00273=-798156,-183832
EC00274=-798156,-183832
EC00275=-798156,-183832
EC00276=-798156,-183832
EC00277=-798156,-183832
EC00278=-798156,-183832
EC00279=-798156,-183832
EC00280=-798156,-183832
EC00281=-798156,-183832
EC00282=-798156,-183832
EC00283=-798156,-183832
EC00284=-798156,-183832
EC00285=-798156,-183832
EC00286=-798156,-183832
EC00287=-798156,-183832
EC00288=-798156,-183832
EC00289=-798156,-183832
EC00290=-798156,-183832
EC00291=-798156,-183832
EC00292=-798156,-183832
EC00293=-798156,-183832
EC00294=-798156,-183832
EC00295=-798156,-183832
EC00296=-798156,-183832
EC00297=-798156,-183832
EC00298=-798156,-183832
EC00299=-798156,-183832
EC00300=-798156,-183832
EC00301=-798156,-183832
EC00302=-798156,-183832
EC00303=-798156,-183832
EC00304=-798156,-183832
EC00305=-798156,-183832
EC00306=-798156,-183832
EC00307=-798156,-183832
EC00308=-798156,-183832
EC00309=-798156,-183832
EC00310=-798156,-183832
EC00311=-798156,-183832
EC00312=-798156,-183832
EC00313=-798156,-183832
EC00314=-798156,-183832
EC00315=-798156,-183832
EC00316=-798156,-183832
EC00317=-798156,-183832
EC00318=-798156,-183832
EC00319=-798156,-183832
EC00320=-798156,-183832
EC00321=-798156,-183832
EC00322=-798156,-183832
EC00323=-798156,-183832
EC00324=-798156,-183832
EC00325=-798156,-183832
EC00326=-798156,-183832
EC00327=-798156,-183832
EC00328=-798156,-183832
EC00329=-798156,-183832
EC00330=-798156,-183832
EC00331=-798156,-183832
EC00332=-798156,-183832
EC00333=-798156,-183832
EC00334=-798156,-183832
EC00335=-798156,-183832
EC00336=-798156,-183832
EC00337=-798156,-183832
EC00338=-798156,-183832
EC00339=-798156,-183832
EC00340=-798156,-183832
EC00341=-798156,-183832
EC00342=-798156,-183832
EC00343=-798156,-183832
EC00344=-798156,-183832
EC00345=-798156,-183832
EC00346=-798156,-183832
EC00347=-798156,-183832
EC00348=-798156,-183832
EC00349=-798156,-183832
EC00350=-798156,-183832
EC00351=-798156,-183832
EC00352=-798156,-183832
EC00353=-798156,-183832
EC00354=-798156,-183832
EC00355=-798156,-183832
EC00356=-798156,-183832
EC00357=-798156,-183832
EC00358=-798156,-183832
///POSTYPE BASE
///RECTAN
///RCONF 0,0,0,0,1,0,0,0,0,0,0,0,0,0,0,0,0,0,0,0,0,0,0,0
P00006=2.006,1.622,-0.565,0.0000,0.0000,0.0000
P00021=0.073,2.058,-0.109,0.0000,0.0000,0.0000
P00022=2.006,1.622,-0.565,0.0000,0.0000,0.0000
///RCONF 0,0,0,0,0,0,0,0,0,0,0,0,0,0,0,0,0,0,0,0,0,0,0,0
P00023=-2.957,-4.083,2.762,0.0000,0.0000,0.0000
P00030=-0.014,-0.768,0.131,0.0000,0.0000,0.0000
P00031=-0.170,0.039,-0.647,0.0000,0.0000,0.0000
P00032=-0.423,0.157,3.222,0.0000,0.0000,0.0000
P00033=0.854,-1.099,3.047,0.0000,0.0000,0.0000
///RCONF 0,0,0,0,1,0,0,0,0,0,0,0,0,0,0,0,0,0,0,0,0,0,0,0
P00034=-8.151,9.743,-4.393,0.0000,0.0000,0.0000
///RCONF 0,0,0,0,0,0,0,0,0,0,0,0,0,0,0,0,0,0,0,0,0,0,0,0
P00035=0.390,-0.027,1.040,0.0000,0.0000,0.0000
P00036=-2.434,0.084,0.197,0.0000,0.0000,0.0000
P00037=-1.075,5.090,-3.949,0.0000,0.0000,0.0000
P00038=0.174,-1.527,-10.860,0.0000,0.0000,0.0000
P00039=-0.109,1.838,-0.266,0.0000,0.0000,0.0000
P00040=2.716,-0.016,3.014,0.0000,0.0000,0.0000
P00041=-0.109,0.014,0.966,0.0000,0.0000,0.0000
P00042=-0.220,0.371,-0.613,0.0000,0.0000,0.0000
P00043=-0.179,-5.890,-3.227,0.0000,0.0000,0.0000
P00044=-8.560,-7.557,-5.232,0.0000,0.0000,0.0000
//INST
///DATE 2024/11/18 22:54
///ATTR SC,RW
///GROUP1 RB1,BS1
///GROUP2 ST1
NOP
'OK_r2_O38-47,64(2)(90,0)
'Down
MOVJ C00000 BC00000 VJ=100.00  +MOVJ EC00000 VJ=100.00
MOVJ C00001 BC00001 VJ=30.00  +MOVJ EC00001 VJ=100.00
'Path S1701
SFTOF3D
MOVJ C00002 BC00002 VJ=50.00  +MOVJ EC00002 VJ=100.00
MOVL C00003 BC00003 V=400.0  +MOVJ EC00003 VJ=100.00
SMOVL C00004 BC00004 V=100.0  +MOVJ EC00004
SREFP 3 C00005 BC00005  +REFP EC00005
CALL JOB:SEARCH-R1-S13D
SET P021 P006
SFTON3D P021
SMOVL C00006 BC00006 V=100.0  +MOVJ EC00006
SMOVL C00007 BC00007 V=100.0  +MOVJ EC00007
SMOVL C00008 BC00008 V=100.0  +MOVJ EC00008
SREFP 3 C00009 BC00009  +REFP EC00009
CALL JOB:SEARCH-R1-S13D
SET P021 P006
SFTON3D P021
SMOVL C00010 BC00010 V=100.0  +MOVJ EC00010
SFTOF3D
SMOVL C00011 BC00011 V=100.0  +MOVJ EC00011
MOVL C00012 BC00012 V=400.0  +MOVJ EC00012 VJ=100.00
MOVL C00013 BC00013 V=1000.0  +MOVJ EC00013 VJ=100.00
MOVJ C00014 BC00014 VJ=100.00  +MOVJ EC00014 VJ=100.00
MOVJ C00015 BC00015 VJ=100.00  +MOVJ EC00015 VJ=100.00
MOVJ C00016 BC00016 VJ=100.00  +MOVJ EC00016 VJ=100.00
MOVJ C00017 BC00017 VJ=100.00  +MOVJ EC00017 VJ=100.00
'Path S1702
SFTOF3D
MOVJ C00018 BC00018 VJ=100.00  +MOVJ EC00018 VJ=100.00
MOVL C00019 BC00019 V=166.7  +MOVJ EC00019 VJ=100.00
SMOVL C00020 BC00020 V=166.7  +MOVJ EC00020
SREFP 3 C00021 BC00021  +REFP EC00021
CALL JOB:SEARCH-R1-S13D
SET P022 P006
SFTON3D P022
SMOVL C00022 BC00022 V=100.0  +MOVJ EC00022
SMOVL C00023 BC00023 V=100.0  +MOVJ EC00023
SMOVL C00024 BC00024 V=100.0  +MOVJ EC00024
SREFP 3 C00025 BC00025  +REFP EC00025
CALL JOB:SEARCH-R1-S13D
SET P022 P006
SFTON3D P022
SMOVL C00026 BC00026 V=100.0  +MOVJ EC00026
SMOVL C00027 BC00027 V=250.0  +MOVJ EC00027
MOVL C00028 BC00028 V=1000.0  +MOVJ EC00028 VJ=100.00
MOVJ C00029 BC00029 VJ=100.00  +MOVJ EC00029 VJ=100.00
'Path S1703
SFTOF3D
MOVJ C00030 BC00030 VJ=100.00  +MOVJ EC00030 VJ=100.00
SMOVL C00031 BC00031 V=250.0  +MOVJ EC00031
SMOVL C00032 BC00032 V=100.0  +MOVJ EC00032
SREFP 3 C00033 BC00033  +REFP EC00033
CALL JOB:SEARCH-R1-S13D
SET P023 P006
SFTON3D P023
SMOVL C00034 BC00034 V=100.0  +MOVJ EC00034
SMOVL C00035 BC00035 V=100.0  +MOVJ EC00035
SMOVL C00036 BC00036 V=100.0  +MOVJ EC00036
SREFP 3 C00037 BC00037  +REFP EC00037
CALL JOB:SEARCH-R1-S13D
SET P023 P006
SFTON3D P023
SMOVL C00038 BC00038 V=166.7  +MOVJ EC00038
SFTOF3D
MOVL C00039 BC00039 V=1000.0  +MOVJ EC00039 VJ=100.00
MOVL C00040 BC00040 V=1000.0  +MOVJ EC00040 VJ=100.00
MOVJ C00041 BC00041 VJ=100.00  +MOVJ EC00041 VJ=100.00
MOVJ C00042 BC00042 VJ=100.00  +MOVJ EC00042 VJ=100.00
MOVJ C00043 BC00043 VJ=100.00  +MOVJ EC00043 VJ=100.00
MOVJ C00044 BC00044 VJ=100.00  +MOVJ EC00044 VJ=100.00
'Up
'Path S1246
SFTOF3D
MOVJ C00045 BC00045 VJ=100.00  +MOVJ EC00045 VJ=100.00
SMOVL C00046 BC00046 V=100.0  +MOVJ EC00046
SREFP 3 C00047 BC00047  +REFP EC00047
CALL JOB:SEARCH-R1-S13D
SET P030 P006
SFTON3D P030
SMOVL C00048 BC00048 V=100.0  +MOVJ EC00048
SREFP 3 C00049 BC00049  +REFP EC00049
CALL JOB:SEARCH-R1-S13D
SET P030 P006
SFTON3D P030
SMOVL C00050 BC00050 V=133.3  +MOVJ EC00050
SFTOF3D
MOVL C00051 BC00051 V=400.0  +MOVJ EC00051 VJ=100.00
SMOVL C00052 BC00052 V=100.0  +MOVJ EC00052
SREFP 3 C00053 BC00053  +REFP EC00053
CALL JOB:SEARCH-R1-S13D
SET P031 P006
SFTON3D P031
SMOVL C00054 BC00054 V=100.0  +MOVJ EC00054
SREFP 3 C00055 BC00055  +REFP EC00055
CALL JOB:SEARCH-R1-S13D
SET P031 P006
SFTON3D P031
SMOVL C00056 BC00056 V=133.3  +MOVJ EC00056
MOVL C00057 BC00057 V=1000.0  +MOVJ EC00057 VJ=100.00
'Path S1276
SFTOF3D
MOVJ C00058 BC00058 VJ=100.00  +MOVJ EC00058 VJ=100.00
MOVL C00059 BC00059 V=400.0  +MOVJ EC00059 VJ=100.00
SMOVL C00060 BC00060 V=100.0  +MOVJ EC00060
SREFP 3 C00061 BC00061  +REFP EC00061
CALL JOB:SEARCH-R1-S13D
SET P032 P006
SFTON3D P032
SMOVL C00062 BC00062 V=100.0  +MOVJ EC00062
SREFP 3 C00063 BC00063  +REFP EC00063
CALL JOB:SEARCH-R1-S13D
SET P032 P006
SFTON3D P032
SMOVL C00064 BC00064 V=100.0  +MOVJ EC00064
MOVL C00065 BC00065 V=400.0  +MOVJ EC00065 VJ=100.00
SFTOF3D
MOVJ C00066 BC00066 VJ=100.00  +MOVJ EC00066 VJ=100.00
SMOVL C00067 BC00067 V=100.0  +MOVJ EC00067
SREFP 3 C00068 BC00068  +REFP EC00068
CALL JOB:SEARCH-R1-S13D
SET P033 P006
SFTON3D P033
SMOVL C00069 BC00069 V=100.0  +MOVJ EC00069
SREFP 3 C00070 BC00070  +REFP EC00070
CALL JOB:SEARCH-R1-S13D
SET P033 P006
SFTON3D P033
SMOVL C00071 BC00071 V=100.0  +MOVJ EC00071
SFTOF3D
MOVL C00072 BC00072 V=400.0  +MOVJ EC00072 VJ=100.00
MOVJ C00073 BC00073 VJ=100.00  +MOVJ EC00073 VJ=100.00
SMOVL C00074 BC00074 V=100.0  +MOVJ EC00074
SREFP 3 C00075 BC00075  +REFP EC00075
CALL JOB:SEARCH-R1-S13D
SET P034 P006
SFTON3D P034
SMOVL C00076 BC00076 V=100.0  +MOVJ EC00076
SREFP 3 C00077 BC00077  +REFP EC00077
CALL JOB:SEARCH-R1-S13D
SET P034 P006
SFTON3D P034
SMOVL C00078 BC00078 V=100.0  +MOVJ EC00078
MOVL C00079 BC00079 V=400.0  +MOVJ EC00079 VJ=100.00
MOVJ C00080 BC00080 VJ=100.00  +MOVJ EC00080 VJ=100.00
'Path S1278
SFTOF3D
MOVJ C00081 BC00081 VJ=100.00  +MOVJ EC00081 VJ=100.00
SMOVL C00082 BC00082 V=100.0  +MOVJ EC00082
SREFP 3 C00083 BC00083  +REFP EC00083
CALL JOB:SEARCH-R1-S13D
SET P035 P006
SFTON3D P035
SMOVL C00084 BC00084 V=100.0  +MOVJ EC00084
SREFP 3 C00085 BC00085  +REFP EC00085
CALL JOB:SEARCH-R1-S13D
SET P035 P006
SFTON3D P035
SMOVL C00086 BC00086 V=100.0  +MOVJ EC00086
SFTOF3D
MOVL C00087 BC00087 V=400.0  +MOVJ EC00087 VJ=100.00
SMOVL C00088 BC00088 V=100.0  +MOVJ EC00088
SREFP 3 C00089 BC00089  +REFP EC00089
CALL JOB:SEARCH-R1-S13D
SET P036 P006
SFTON3D P036
SMOVL C00090 BC00090 V=100.0  +MOVJ EC00090
SREFP 3 C00091 BC00091  +REFP EC00091
CALL JOB:SEARCH-R1-S13D
SET P036 P006
SFTON3D P036
SMOVL C00092 BC00092 V=100.0  +MOVJ EC00092
'Path S1970
SFTOF3D
MOVJ C00093 BC00093 VJ=100.00  +MOVJ EC00093 VJ=100.00
MOVL C00094 BC00094 V=400.0  +MOVJ EC00094 VJ=100.00
SMOVL C00095 BC00095 V=100.0  +MOVJ EC00095
SREFP 3 C00096 BC00096  +REFP EC00096
CALL JOB:SEARCH-R1-S13D
SET P037 P006
SFTON3D P037
SMOVL C00097 BC00097 V=100.0  +MOVJ EC00097
SREFP 3 C00098 BC00098  +REFP EC00098
CALL JOB:SEARCH-R1-S13D
SET P037 P006
SFTON3D P037
SMOVL C00099 BC00099 V=100.0  +MOVJ EC00099
SFTOF3D
MOVL C00100 BC00100 V=400.0  +MOVJ EC00100 VJ=100.00
MOVL C00101 BC00101 V=1000.0  +MOVJ EC00101 VJ=100.00
MOVJ C00102 BC00102 VJ=100.00  +MOVJ EC00102 VJ=100.00
SMOVL C00103 BC00103 V=100.0  +MOVJ EC00103
SREFP 3 C00104 BC00104  +REFP EC00104
CALL JOB:SEARCH-R1-S13D
SET P038 P006
SFTON3D P038
SMOVL C00105 BC00105 V=100.0  +MOVJ EC00105
SREFP 3 C00106 BC00106  +REFP EC00106
CALL JOB:SEARCH-R1-S13D
SET P038 P006
SFTON3D P038
SMOVL C00107 BC00107 V=100.0  +MOVJ EC00107
SFTOF3D
MOVL C00108 BC00108 V=400.0  +MOVJ EC00108 VJ=100.00
SMOVL C00109 BC00109 V=100.0  +MOVJ EC00109
SREFP 3 C00110 BC00110  +REFP EC00110
CALL JOB:SEARCH-R1-S13D
SET P039 P006
SFTON3D P039
SMOVL C00111 BC00111 V=100.0  +MOVJ EC00111
SREFP 3 C00112 BC00112  +REFP EC00112
CALL JOB:SEARCH-R1-S13D
SET P039 P006
SFTON3D P039
SMOVL C00113 BC00113 V=100.0  +MOVJ EC00113
MOVJ C00114 BC00114 VJ=100.00  +MOVJ EC00114 VJ=100.00
SFTOF3D
MOVJ C00115 BC00115 VJ=100.00  +MOVJ EC00115 VJ=100.00
MOVJ C00116 BC00116 VJ=100.00  +MOVJ EC00116 VJ=100.00
MOVJ C00117 BC00117 VJ=100.00  +MOVJ EC00117 VJ=100.00
MOVJ C00118 BC00118 VJ=100.00  +MOVJ EC00118 VJ=100.00
SMOVL C00119 BC00119 V=100.0  +MOVJ EC00119
SREFP 3 C00120 BC00120  +REFP EC00120
CALL JOB:SEARCH-R1-S13D
SET P040 P006
SFTON3D P040
SMOVL C00121 BC00121 V=100.0  +MOVJ EC00121
SREFP 3 C00122 BC00122  +REFP EC00122
CALL JOB:SEARCH-R1-S13D
SET P040 P006
SFTON3D P040
SMOVL C00123 BC00123 V=100.0  +MOVJ EC00123
SFTOF3D
MOVL C00124 BC00124 V=1000.0  +MOVJ EC00124 VJ=100.00
SMOVL C00125 BC00125 V=100.0  +MOVJ EC00125
SREFP 3 C00126 BC00126  +REFP EC00126
CALL JOB:SEARCH-R1-S13D
SET P041 P006
SFTON3D P041
SMOVL C00127 BC00127 V=100.0  +MOVJ EC00127
SREFP 3 C00128 BC00128  +REFP EC00128
CALL JOB:SEARCH-R1-S13D
SET P041 P006
SFTON3D P041
SMOVL C00129 BC00129 V=100.0  +MOVJ EC00129
MOVJ C00130 BC00130 VJ=100.00  +MOVJ EC00130 VJ=100.00
SFTOF3D
MOVJ C00131 BC00131 VJ=100.00  +MOVJ EC00131 VJ=100.00
MOVL C00132 BC00132 V=400.0  +MOVJ EC00132 VJ=100.00
SMOVL C00133 BC00133 V=100.0  +MOVJ EC00133
SREFP 3 C00134 BC00134  +REFP EC00134
CALL JOB:SEARCH-R1-S13D
SET P042 P006
SFTON3D P042
SMOVL C00135 BC00135 V=100.0  +MOVJ EC00135
SREFP 3 C00136 BC00136  +REFP EC00136
CALL JOB:SEARCH-R1-S13D
SET P042 P006
SFTON3D P042
SMOVL C00137 BC00137 V=100.0  +MOVJ EC00137
SFTOF3D
MOVL C00138 BC00138 V=400.0  +MOVJ EC00138 VJ=100.00
'Path S1282
SFTOF3D
SMOVL C00139 BC00139 V=100.0  +MOVJ EC00139
SREFP 3 C00140 BC00140  +REFP EC00140
CALL JOB:SEARCH-R1-S13D
SET P043 P006
SFTON3D P043
SMOVL C00141 BC00141 V=100.0  +MOVJ EC00141
SREFP 3 C00142 BC00142  +REFP EC00142
CALL JOB:SEARCH-R1-S13D
SET P043 P006
SFTON3D P043
SMOVL C00143 BC00143 V=100.0  +MOVJ EC00143
SFTOF3D
MOVL C00144 BC00144 V=400.0  +MOVJ EC00144 VJ=100.00
MOVL C00145 BC00145 V=1000.0  +MOVJ EC00145 VJ=100.00
MOVJ C00146 BC00146 VJ=100.00  +MOVJ EC00146 VJ=100.00
MOVJ C00147 BC00147 VJ=100.00  +MOVJ EC00147 VJ=100.00
MOVL C00148 BC00148 V=400.0  +MOVJ EC00148 VJ=100.00
SMOVL C00149 BC00149 V=100.0  +MOVJ EC00149
SREFP 3 C00150 BC00150  +REFP EC00150
CALL JOB:SEARCH-R1-S13D
SET P044 P006
SFTON3D P044
SMOVL C00151 BC00151 V=100.0  +MOVJ EC00151
SREFP 3 C00152 BC00152  +REFP EC00152
CALL JOB:SEARCH-R1-S13D
SET P044 P006
SFTON3D P044
SMOVL C00153 BC00153 V=100.0  +MOVJ EC00153
MOVL C00154 BC00154 V=400.0  +MOVJ EC00154 VJ=100.00
SFTON3D P044
SMOVL C00155 BC00155 V=133.3 PL=0  +MOVJ EC00155
SREFP 1 C00156 BC00156  +REFP EC00156
SREFP 2 C00157 BC00157  +REFP EC00157
MACRO1 MJ#(0) ARGF9
ARCON
SWVON WEV#(60)
SMOVL C00158 BC00158 V=8.3  +MOVJ EC00158
SMOVL C00159 BC00159 V=8.3  +MOVJ EC00159
SMOVL C00160 BC00160 V=8.3  +MOVJ EC00160
ARCOF
SWVOF
SMOVL C00161 BC00161 V=250.0  +MOVJ EC00161
SFTOF3D
MOVJ C00162 BC00162 VJ=100.00  +MOVJ EC00162 VJ=100.00
SFTOF3D
MOVJ C00163 BC00163 VJ=70.00  +MOVJ EC00163 VJ=100.00
'Path W1138
MOVJ C00164 BC00164 VJ=100.00  +MOVJ EC00164 VJ=100.00
SFTOF
SFTON3D P037
SMOVL C00165 BC00165 V=133.3 PL=0  +MOVJ EC00165
SREFP 1 C00166 BC00166  +REFP EC00166
SREFP 2 C00167 BC00167  +REFP EC00167
MACRO1 MJ#(0) ARGF9
ARCON
SWVON WEV#(60)
SMOVL C00168 BC00168 V=8.3  +MOVJ EC00168
SMOVL C00169 BC00169 V=8.3  +MOVJ EC00169
SMOVL C00170 BC00170 V=8.3  +MOVJ EC00170
ARCOF
SWVOF
SMOVL C00171 BC00171 V=400.0  +MOVJ EC00171
MOVJ C00172 BC00172 VJ=100.00  +MOVJ EC00172 VJ=100.00
SFTOF3D
MOVJ C00173 BC00173 VJ=100.00  +MOVJ EC00173 VJ=100.00
MOVJ C00174 BC00174 VJ=100.00  +MOVJ EC00174 VJ=100.00
SFTON3D P039
SMOVL C00175 BC00175 V=133.3 PL=0  +MOVJ EC00175
SREFP 1 C00176 BC00176  +REFP EC00176
SREFP 2 C00177 BC00177  +REFP EC00177
MACRO1 MJ#(0) ARGF14
ARCON
SFTON3D P038
SMOVL C00178 BC00178 V=8.3  +MOVJ EC00178
SMOVL C00179 BC00179 V=8.3  +MOVJ EC00179
ARCOF
SMOVL C00180 BC00180 V=400.0  +MOVJ EC00180
SFTOF3D
MOVJ C00181 BC00181 VJ=100.00  +MOVJ EC00181 VJ=100.00
MOVJ C00182 BC00182 VJ=100.00  +MOVJ EC00182 VJ=100.00
MOVJ C00183 BC00183 VJ=100.00  +MOVJ EC00183 VJ=100.00
MOVJ C00184 BC00184 VJ=100.00  +MOVJ EC00184 VJ=100.00
'Path W1140
SFTOF3D
SFTON3D P033
SMOVL C00185 BC00185 V=133.3 PL=0  +MOVJ EC00185
SREFP 1 C00186 BC00186  +REFP EC00186
SREFP 2 C00187 BC00187  +REFP EC00187
MACRO1 MJ#(0) ARGF14
ARCON
SWVON WEV#(10)
SMOVL C00188 BC00188 V=8.3  +MOVJ EC00188
SFTON3D P032
SMOVL C00189 BC00189 V=8.3  +MOVJ EC00189
SMOVL C00190 BC00190 V=8.3  +MOVJ EC00190
ARCOF
SWVOF
SMOVL C00191 BC00191 V=400.0  +MOVJ EC00191
SFTOF3D
MOVJ C00192 BC00192 VJ=100.00  +MOVJ EC00192 VJ=100.00
SFTOF3D
MOVJ C00193 BC00193 VJ=100.00  +MOVJ EC00193 VJ=100.00
'Path W1142
SFTOF3D
SFTON3D P030
MOVJ C00194 BC00194 VJ=100.00  +MOVJ EC00194 VJ=100.00
SMOVL C00195 BC00195 V=133.3 PL=0  +MOVJ EC00195
SREFP 1 C00196 BC00196  +REFP EC00196
SREFP 2 C00197 BC00197  +REFP EC00197
MACRO1 MJ#(0) ARGF9
ARCON
SMOVL C00198 BC00198 V=8.3  +MOVJ EC00198
SFTON3D P031
SMOVL C00199 BC00199 V=8.3  +MOVJ EC00199
SMOVL C00200 BC00200 V=8.3  +MOVJ EC00200
SMOVL C00201 BC00201 V=8.3  +MOVJ EC00201
ARCOF
SMOVL C00202 BC00202 V=400.0  +MOVJ EC00202
SFTOF3D
MOVJ C00203 BC00203 VJ=100.00  +MOVJ EC00203 VJ=100.00
'Path W1143
SFTOF3D
SFTON3D P034
MOVJ C00204 BC00204 VJ=100.00  +MOVJ EC00204 VJ=100.00
SMOVL C00205 BC00205 V=133.3 PL=0  +MOVJ EC00205
SREFP 1 C00206 BC00206  +REFP EC00206
SREFP 2 C00207 BC00207  +REFP EC00207
MACRO1 MJ#(0) ARGF9
ARCON
SMOVC C00208 BC00208 V=8.3  +MOVJ EC00208
SMOVC C00209 BC00209 V=8.3  +MOVJ EC00209
SMOVC C00210 BC00210 V=8.3  +MOVJ EC00210
SMOVL C00211 BC00211 V=8.3  +MOVJ EC00211
SMOVC C00212 BC00212 V=8.3  +MOVJ EC00212
SMOVC C00213 BC00213 V=8.3  +MOVJ EC00213
SMOVC C00214 BC00214 V=8.3  +MOVJ EC00214
ARCOF
SMOVL C00215 BC00215 V=400.0  +MOVJ EC00215
SFTOF3D
MOVJ C00216 BC00216 VJ=100.00  +MOVJ EC00216 VJ=100.00
'Path W1144
SFTOF3D
SFTON3D P036
MOVJ C00217 BC00217 VJ=100.00  +MOVJ EC00217 VJ=100.00
SFTON3D P036
SMOVL C00218 BC00218 V=133.3 PL=0  +MOVJ EC00218
SREFP 1 C00219 BC00219  +REFP EC00219
SREFP 2 C00220 BC00220  +REFP EC00220
MACRO1 MJ#(0) ARGF14
ARCON
SMOVL C00221 BC00221 V=9.2  +MOVJ EC00221
SFTON3D P035
SMOVL C00222 BC00222 V=9.2  +MOVJ EC00222
SMOVL C00223 BC00223 V=9.2  +MOVJ EC00223
ARCOF
SMOVL C00224 BC00224 V=400.0  +MOVJ EC00224
SFTOF3D
MOVJ C00225 BC00225 VJ=100.00  +MOVJ EC00225 VJ=100.00
MOVJ C00226 BC00226 VJ=100.00  +MOVJ EC00226 VJ=100.00
SFTON3D P042
SMOVL C00227 BC00227 V=133.3 PL=0  +MOVJ EC00227
SREFP 1 C00228 BC00228  +REFP EC00228
SREFP 2 C00229 BC00229  +REFP EC00229
MACRO1 MJ#(0) ARGF14
ARCON
SMOVL C00230 BC00230 V=10.0  +MOVJ EC00230
SFTON3D P043
SMOVL C00231 BC00231 V=10.0  +MOVJ EC00231
SMOVL C00232 BC00232 V=10.0  +MOVJ EC00232
ARCOF
SMOVL C00233 BC00233 V=400.0  +MOVJ EC00233
MOVJ C00234 BC00234 VJ=100.00  +MOVJ EC00234 VJ=100.00
MOVJ C00235 BC00235 VJ=100.00  +MOVJ EC00235 VJ=100.00
SFTOF3D
SFTON3D P040
SMOVL C00236 BC00236 V=133.3 PL=0  +MOVJ EC00236
SREFP 1 C00237 BC00237  +REFP EC00237
SREFP 2 C00238 BC00238  +REFP EC00238
MACRO1 MJ#(0) ARGF14
ARCON
SMOVL C00239 BC00239 V=10.0  +MOVJ EC00239
SFTON3D P041
SMOVL C00240 BC00240 V=10.0  +MOVJ EC00240
SMOVL C00241 BC00241 V=10.0  +MOVJ EC00241
ARCOF
SMOVL C00242 BC00242 V=400.0  +MOVJ EC00242
SFTOF3D
MOVJ C00243 BC00243 VJ=100.00  +MOVJ EC00243 VJ=100.00
MOVJ C00244 BC00244 VJ=100.00  +MOVJ EC00244 VJ=100.00
MOVJ C00245 BC00245 VJ=100.00  +MOVJ EC00245 VJ=100.00
MOVJ C00246 BC00246 VJ=100.00  +MOVJ EC00246 VJ=100.00
MOVJ C00247 BC00247 VJ=100.00  +MOVJ EC00247 VJ=100.00
'Down
'1
MOVJ C00248 BC00248 VJ=100.00  +MOVJ EC00248 VJ=100.00
'Path W1705
SFTOF3D
SFTON3D P023
MOVJ C00249 BC00249 VJ=100.00  +MOVJ EC00249 VJ=100.00
SMOVL C00250 BC00250 V=400.0  +MOVJ EC00250
SMOVL C00251 BC00251 V=133.3 PL=0  +MOVJ EC00251
SREFP 1 C00252 BC00252  +REFP EC00252
SREFP 2 C00253 BC00253  +REFP EC00253
MACRO1 MJ#(0) ARGF14
ARCON
SMOVL C00254 BC00254 V=10.0  +MOVJ EC00254
ARCOF
SMOVL C00255 BC00255 V=400.0  +MOVJ EC00255
SMOVL C00256 BC00256 V=1000.0  +MOVJ EC00256
SFTOF3D
MOVJ C00257 BC00257 VJ=100.00  +MOVJ EC00257 VJ=100.00
MOVJ C00258 BC00258 VJ=100.00  +MOVJ EC00258 VJ=100.00
'2
MOVJ C00259 BC00259 VJ=100.00  +MOVJ EC00259 VJ=100.00
MOVJ C00260 BC00260 VJ=100.00  +MOVJ EC00260 VJ=100.00
MOVJ C00261 BC00261 VJ=100.00  +MOVJ EC00261 VJ=100.00
'Path W1706
SFTOF3D
SFTON3D P021
MOVJ C00262 BC00262 VJ=15.00  +MOVJ EC00262 VJ=100.00
SMOVL C00263 BC00263 V=400.0  +MOVJ EC00263
SMOVL C00264 BC00264 V=100.0 PL=0  +MOVJ EC00264
SREFP 1 C00265 BC00265  +REFP EC00265
SREFP 2 C00266 BC00266  +REFP EC00266
MACRO1 MJ#(0) ARGF14
ARCON
SMOVL C00267 BC00267 V=10.0  +MOVJ EC00267
ARCOF
SMOVL C00268 BC00268 V=166.7  +MOVJ EC00268
SMOVL C00269 BC00269 V=166.7  +MOVJ EC00269
SMOVL C00270 BC00270 V=166.7  +MOVJ EC00270
ARCON
SMOVL C00271 BC00271 V=10.0  +MOVJ EC00271
ARCOF
SMOVL C00272 BC00272 V=166.7  +MOVJ EC00272
SMOVL C00273 BC00273 V=400.0  +MOVJ EC00273
SMOVL C00274 BC00274 V=1000.0  +MOVJ EC00274
SFTOF3D
MOVJ C00275 BC00275 VJ=20.00  +MOVJ EC00275 VJ=20.00
'Path W1707
SFTOF3D
SFTON3D P021
MOVJ C00276 BC00276 VJ=100.00  +MOVJ EC00276 VJ=100.00
SMOVL C00277 BC00277 V=400.0  +MOVJ EC00277
SMOVL C00278 BC00278 V=100.0 PL=0  +MOVJ EC00278
SREFP 1 C00279 BC00279  +REFP EC00279
SREFP 2 C00280 BC00280  +REFP EC00280
MACRO1 MJ#(0) ARGF14
ARCON
SMOVL C00281 BC00281 V=10.0  +MOVJ EC00281
ARCOF
SMOVL C00282 BC00282 V=166.7  +MOVJ EC00282
SMOVL C00283 BC00283 V=166.7  +MOVJ EC00283
SMOVL C00284 BC00284 V=166.7  +MOVJ EC00284
ARCON
SMOVL C00285 BC00285 V=10.0  +MOVJ EC00285
ARCOF
SMOVL C00286 BC00286 V=400.0  +MOVJ EC00286
SMOVL C00287 BC00287 V=1000.0  +MOVJ EC00287
SFTOF3D
MOVJ C00288 BC00288 VJ=100.00  +MOVJ EC00288 VJ=100.00
MOVJ C00289 BC00289 VJ=100.00  +MOVJ EC00289 VJ=100.00
'3
MOVJ C00290 BC00290 VJ=100.00  +MOVJ EC00290 VJ=100.00
MOVJ C00291 BC00291 VJ=100.00  +MOVJ EC00291 VJ=100.00
'Path W1709
SFTOF3D
SFTON3D P023
MOVJ C00292 BC00292 VJ=100.00  +MOVJ EC00292 VJ=100.00
SMOVL C00293 BC00293 V=400.0  +MOVJ EC00293
SMOVL C00294 BC00294 V=133.3 PL=0  +MOVJ EC00294
SREFP 1 C00295 BC00295  +REFP EC00295
SREFP 2 C00296 BC00296  +REFP EC00296
MACRO1 MJ#(0) ARGF14
ARCON
SMOVL C00297 BC00297 V=10.0  +MOVJ EC00297
ARCOF
SMOVL C00298 BC00298 V=400.0  +MOVJ EC00298
SMOVL C00299 BC00299 V=1000.0  +MOVJ EC00299
SFTOF3D
MOVJ C00300 BC00300 VJ=100.00  +MOVJ EC00300 VJ=100.00
MOVJ C00301 BC00301 VJ=100.00  +MOVJ EC00301 VJ=100.00
'4
MOVJ C00302 BC00302 VJ=100.00  +MOVJ EC00302 VJ=100.00
MOVJ C00303 BC00303 VJ=100.00  +MOVJ EC00303 VJ=100.00
'Path W1710
SFTOF3D
SFTON3D P021
MOVJ C00304 BC00304 VJ=15.00  +MOVJ EC00304 VJ=100.00
SMOVL C00305 BC00305 V=400.0  +MOVJ EC00305
SMOVL C00306 BC00306 V=133.3 PL=0  +MOVJ EC00306
SREFP 1 C00307 BC00307  +REFP EC00307
SREFP 2 C00308 BC00308  +REFP EC00308
MACRO1 MJ#(0) ARGF14
ARCON
SMOVL C00309 BC00309 V=10.0  +MOVJ EC00309
ARCOF
SMOVL C00310 BC00310 V=400.0  +MOVJ EC00310
SMOVL C00311 BC00311 V=1000.0  +MOVJ EC00311
SFTOF3D
'Path W1711
SFTOF3D
SFTON3D P021
MOVJ C00312 BC00312 VJ=100.00  +MOVJ EC00312 VJ=100.00
SMOVL C00313 BC00313 V=400.0  +MOVJ EC00313
SMOVL C00314 BC00314 V=133.3 PL=0  +MOVJ EC00314
SREFP 1 C00315 BC00315  +REFP EC00315
SREFP 2 C00316 BC00316  +REFP EC00316
MACRO1 MJ#(0) ARGF14
ARCON
SMOVL C00317 BC00317 V=10.0  +MOVJ EC00317
ARCOF
SMOVL C00318 BC00318 V=400.0  +MOVJ EC00318
SMOVL C00319 BC00319 V=1000.0  +MOVJ EC00319
SFTOF3D
MOVJ C00320 BC00320 VJ=100.00  +MOVJ EC00320 VJ=100.00
MOVJ C00321 BC00321 VJ=100.00  +MOVJ EC00321 VJ=100.00
'6
MOVJ C00322 BC00322 VJ=100.00  +MOVJ EC00322 VJ=100.00
MOVJ C00323 BC00323 VJ=100.00  +MOVJ EC00323 VJ=100.00
'Path W1714
SFTOF3D
SFTON3D P022
MOVJ C00324 BC00324 VJ=100.00  +MOVJ EC00324 VJ=100.00
MOVJ C00325 BC00325 VJ=20.00  +MOVJ EC00325 VJ=20.00
SMOVL C00326 BC00326 V=400.0  +MOVJ EC00326
SMOVL C00327 BC00327 V=133.3 PL=0  +MOVJ EC00327
SREFP 1 C00328 BC00328  +REFP EC00328
SREFP 2 C00329 BC00329  +REFP EC00329
MACRO1 MJ#(0) ARGF14
ARCON
SMOVL C00330 BC00330 V=10.0  +MOVJ EC00330
ARCOF
SMOVL C00331 BC00331 V=400.0  +MOVJ EC00331
SMOVL C00332 BC00332 V=1000.0  +MOVJ EC00332
SFTOF3D
'Path W1715
SFTOF3D
SFTON3D P022
MOVJ C00333 BC00333 VJ=100.00  +MOVJ EC00333 VJ=100.00
SMOVL C00334 BC00334 V=400.0  +MOVJ EC00334
SMOVL C00335 BC00335 V=133.3 PL=0  +MOVJ EC00335
SREFP 1 C00336 BC00336  +REFP EC00336
SREFP 2 C00337 BC00337  +REFP EC00337
MACRO1 MJ#(0) ARGF14
ARCON
SMOVL C00338 BC00338 V=10.0  +MOVJ EC00338
ARCOF
SMOVL C00339 BC00339 V=400.0  +MOVJ EC00339
SMOVL C00340 BC00340 V=250.0  +MOVJ EC00340
SMOVL C00341 BC00341 V=166.7  +MOVJ EC00341
ARCON
SMOVL C00342 BC00342 V=10.0  +MOVJ EC00342
ARCOF
SMOVL C00343 BC00343 V=250.0  +MOVJ EC00343
SFTOF3D
MOVJ C00344 BC00344 VJ=100.00  +MOVJ EC00344 VJ=14.00
MOVJ C00345 BC00345 VJ=100.00  +MOVJ EC00345 VJ=100.00
MOVJ C00346 BC00346 VJ=100.00  +MOVJ EC00346 VJ=100.00
MOVJ C00347 BC00347 VJ=100.00  +MOVJ EC00347 VJ=100.00
MOVJ C00348 BC00348 VJ=100.00  +MOVJ EC00348 VJ=100.00
'7
MOVJ C00349 BC00349 VJ=100.00  +MOVJ EC00349 VJ=100.00
'Path W1716
SFTOF3D
SFTON3D P022
MOVJ C00350 BC00350 VJ=100.00  +MOVJ EC00350 VJ=25.00
SMOVL C00351 BC00351 V=400.0  +MOVJ EC00351
SMOVL C00352 BC00352 V=133.3 PL=0  +MOVJ EC00352
SREFP 1 C00353 BC00353  +REFP EC00353
SREFP 2 C00354 BC00354  +REFP EC00354
MACRO1 MJ#(0) ARGF14
ARCON
SMOVL C00355 BC00355 V=11.7  +MOVJ EC00355
ARCOF
SMOVL C00356 BC00356 V=400.0  +MOVJ EC00356
SFTOF3D
MOVJ C00357 BC00357 VJ=50.00  +MOVJ EC00357 VJ=100.00
SMOVL C00358 BC00358 V=1000.0  +MOVJ EC00358
SFTOF3D
END
